FUNCTION_BLOCK UT_SoftkeyMapping_UP (* Service Interface Function Block Type *)
  (* Standard: ISO 11783-6; Classification: Soft Key – ISO 11783-6 – B.6; Function: All Inputs; Type: UT according to ISO 11783-6; Description: this maps to IE *)
  (* Version 1.0, 2018-12-05, Jose Cabral *)
  (* Version 1.1, 2022-08-04, Franz Höpfinger, HR Agrartechnik GmbH *)
  (* Version 1.2, 2023-01-05, Franz Höpfinger, HR Agrartechnik GmbH *)
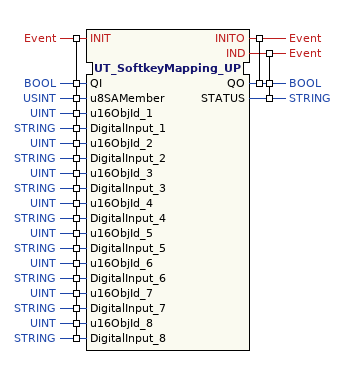
  EVENT_INPUT
    INIT WITH QI, u8SAMember, u16ObjId_1, DigitalInput_1, u16ObjId_2, DigitalInput_2, u16ObjId_3, DigitalInput_3, u16ObjId_4, DigitalInput_4, u16ObjId_5, DigitalInput_5, u16ObjId_6, DigitalInput_6, u16ObjId_7, DigitalInput_7, u16ObjId_8, DigitalInput_8; (* Service Initialization *)
  END_EVENT
  EVENT_OUTPUT
    INITO WITH QO; (* Initialization Confirm *)
    IND WITH QO, STATUS; (* Indication from Resource *)
  END_EVENT
  VAR_INPUT
    QI : BOOL; (* Event Input Qualifier *)
    u8SAMember : USINT := 255; (* Dummy !, set to 255 if in doubt. 0 deactivates FB. *)
    u16ObjId_1 : UINT; (* Object ID of Input 1 *)
    DigitalInput_1 : STRING; (* Identifier for Input 1 *)
    u16ObjId_2 : UINT; (* Object ID of Input 2 *)
    DigitalInput_2 : STRING; (* Identifier for Input 2 *)
    u16ObjId_3 : UINT; (* Object ID of Input 3 *)
    DigitalInput_3 : STRING; (* Identifier for Input 3 *)
    u16ObjId_4 : UINT; (* Object ID of Input 4 *)
    DigitalInput_4 : STRING; (* Identifier for Input 4 *)
    u16ObjId_5 : UINT; (* Object ID of Input 5 *)
    DigitalInput_5 : STRING; (* Identifier for Input 5 *)
    u16ObjId_6 : UINT; (* Object ID of Input 6 *)
    DigitalInput_6 : STRING; (* Identifier for Input 6 *)
    u16ObjId_7 : UINT; (* Object ID of Input 7 *)
    DigitalInput_7 : STRING; (* Identifier for Input 7 *)
    u16ObjId_8 : UINT; (* Object ID of Input 8 *)
    DigitalInput_8 : STRING; (* Identifier for Input 8 *)
  END_VAR
  VAR_OUTPUT
    QO : BOOL; (* Event Output Qualifier *)
    STATUS : STRING; (* Service Status *)
  END_VAR
END_FUNCTION_BLOCK
